{attribute 'GeneratedUsingTerminal: ELX2002-0000-0016'}
{attribute addProperty BoxType "ELX2002-0000-0016"}
{attribute addProperty Id "OutputAT %Q*BOOL1"}
{attribute addProperty CRC "1120571895"}
{attribute addProperty Size "1"}
TYPE Channel_42CA91F7 :
STRUCT
	{attribute addProperty Name "Output"}
	Output AT %Q* : BOOL;
END_STRUCT
END_TYPE

(* stored: Version 1.2.0.0, ProductVersion 3.1.4024.9
   DUT Channel_42CA91F7: Id {9fe2ebf9-0d66-45fd-aa5b-7b19bc09ebf3} *)
